// TIA Portal V17 export
// export: Created 2022-02-03T14:45:12.0016081Z, ExportSetting WithDefaults, DisplayName Totally Integrated Automation Portal, DisplayVersion V17, DisplayName TIA Portal Openness, DisplayVersion V17, DisplayName TIA Portal Version Control Interface, DisplayVersion V17, DisplayName SINAMICS Startdrive Advanced, DisplayVersion V17, DisplayName SINAMICS Startdrive G130, G150, S120, S150, SINAMICS MV, S210, DisplayVersion V17, DisplayName SINAMICS Startdrive G110M, G120, G120C, G120D, G120P, G115D, DisplayVersion V17, DisplayName STEP 7 Professional, DisplayVersion V17, DisplayName STEP 7 Safety, DisplayVersion V17, DisplayName WinCC Advanced, DisplayVersion V17
DATA_BLOCK "lifeBitControl_DB"   // DB9
VERSION : 0.1
// stored: Access Unpublished, AutoNumber true, DBAccessibleFromOPCUA true, DBAccessibleFromWebserver true, InstanceOfName lifeBitControl, InstanceOfType FB
"lifeBitControl"
   // VAR_INPUT
   //    acknowledge : Bool;
   // END_VAR
   // VAR_OUTPUT
   //    warning : Bool;
   // END_VAR
   // VAR
   //    statTPCoordination : Word;
   //    IntIEC_Timer1 { S7_SetPoint := 'True'} : TON_TIME;
   //    InstIEC_Timer2 { S7_SetPoint := 'True'} : TON_TIME;
   //    statOldAcknowledge { S7_SetPoint := 'True'} : Bool;
   //    statOldTimer : Bool;
   // END_VAR
BEGIN
END_DATA_BLOCK
